FUNCTION_BLOCK BaseMemberExternAdd (* Adds an external member to the network list manually. *)
  (* Standard: 61499-2; Description: The use of this function is not ISO 11783 Part 5 conform. \n Use this function only if you must communicate with an external CF, \n that does not send a address claimed message. \n An address claimed message of an external CF with the same source address \n will replace this manual added member entry.  \n The function works independent from the configuration of the #CFG_PARAM_EXTERNAL_ADDR_CLAIM parameter. \n The added CF will be set to announced in the next iso_DlCyclicGlobal() run. *)
  (* Version 1.0, 2026-01-16, Gemini, initial API and implementation and/or initial documentation *)
  PACKAGE isobus::pgn;
  IMPORT eclipse4diac::core::TypeHash;
  IMPORT isobus::pgn::ISO_CAN_NODE::NODE1;
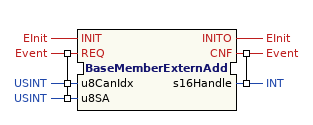
  EVENT_INPUT
    INIT : EInit; (* Service Initialization *)
    REQ WITH u8SA, u8CanIdx; (* Add external member *)
  END_EVENT
  EVENT_OUTPUT
    INITO : EInit; (* Initialization Confirm *)
    CNF WITH s16Handle; (* Confirmation *)
  END_EVENT
  VAR_INPUT
    u8CanIdx : USINT := NODE1; (* CAN node index *)
    u8SA : USINT; (* Source Address of the CF to add *)
  END_VAR
  VAR_OUTPUT
    s16Handle : INT; (* Handle of the added member *)
  END_VAR
END_FUNCTION_BLOCK
